FUNCTION_BLOCK SETTINGSVALIDATOR (* Value validator for setting the parameters of the flotation tank *)
  (* Version 1.0, AN, SWDC RTSoft *)
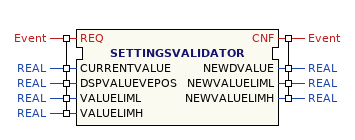
  EVENT_INPUT
    REQ WITH CURRENTVALUE, DSPVALUEVEPOS, VALUELIML, VALUELIMH;
  END_EVENT
  EVENT_OUTPUT
    CNF WITH NEWDVALUE, NEWVALUELIML, NEWVALUELIMH;
  END_EVENT
  VAR_INPUT
    CURRENTVALUE : REAL;
    DSPVALUEVEPOS : REAL;
    VALUELIML : REAL;
    VALUELIMH : REAL;
  END_VAR
  VAR_OUTPUT
    NEWDVALUE : REAL;
    NEWVALUELIML : REAL;
    NEWVALUELIMH : REAL;
  END_VAR
END_FUNCTION_BLOCK
